// TIA Portal V21 export
FUNCTION "STANDARD" : Void   // FC13, LAD
{ S7_Optimized_Access := 'TRUE' }
// stored: SetENOAutomatically false
   VAR_TEMP
      "std temp3 hyst" : Real;
   END_VAR
   VAR_TEMP   // added for the SCL form of the ladder/FBD networks
      _w1 : Bool;
      _w2 : Bool;
      _w3 : Bool;
      _w4 : Bool;
   END_VAR
BEGIN

REGION Network 1
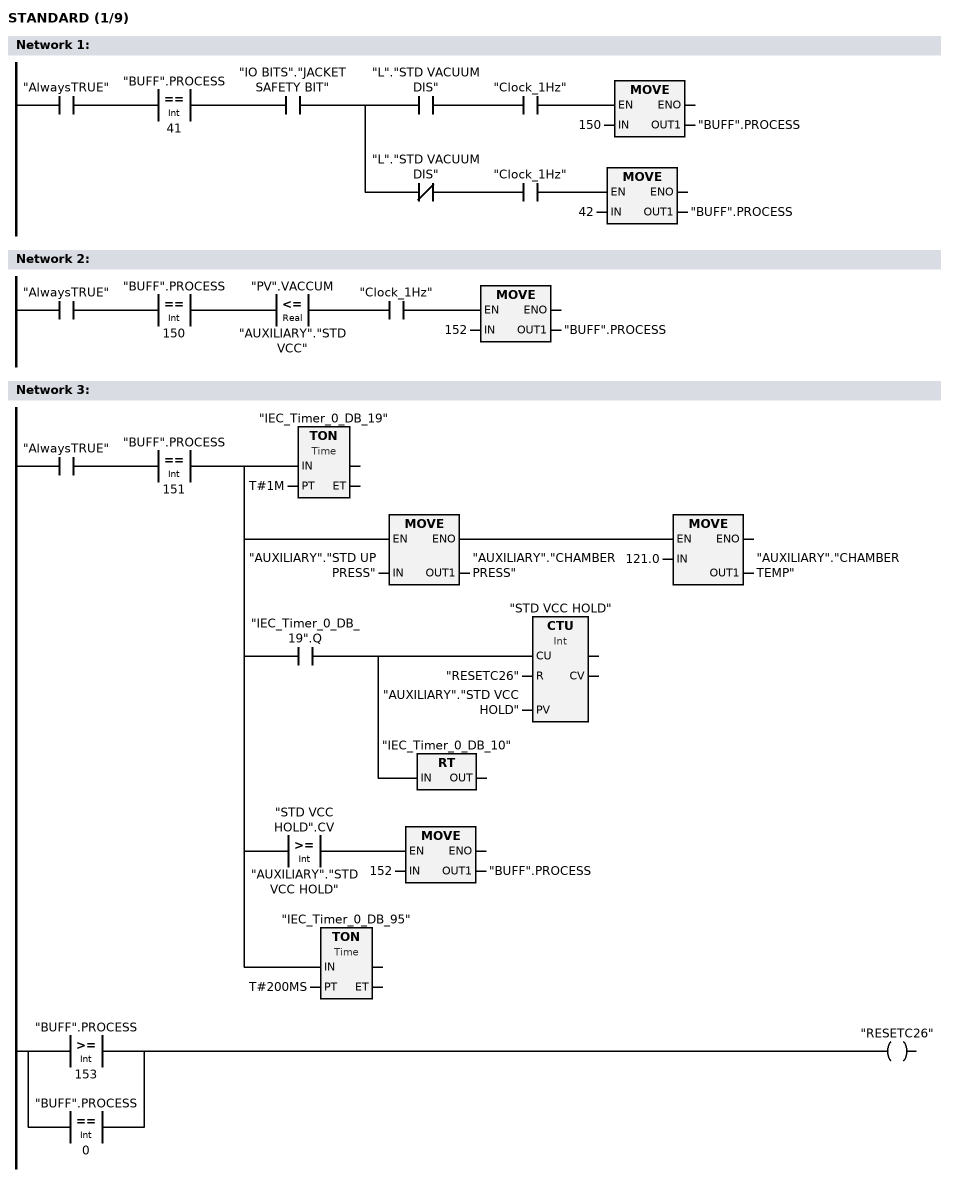
   RUNG wire#powerrail
      Contact( "AlwaysTRUE" )
      { S7_Templates := "SrcType := Int" } EQ_Contact(in1 := "BUFF".PROCESS, in2 := 41)
      Contact( "IO BITS"."JACKET SAFETY BIT" )
      wire#w1
      Contact( "L"."STD VACUUM DIS" )
      Contact( "Clock_1Hz" )
      Move(in := 150, out1 => "BUFF".PROCESS)
   END_RUNG
   RUNG wire#w1
      I_Contact( "L"."STD VACUUM DIS" )
      Contact( "Clock_1Hz" )
      Move(in := 42, out1 => "BUFF".PROCESS)
   END_RUNG
   // the same network as SCL:
   #_w1 := "AlwaysTRUE" AND ("BUFF".PROCESS = 41) AND "IO BITS"."JACKET SAFETY BIT";
   IF #_w1 AND "L"."STD VACUUM DIS" AND "Clock_1Hz" THEN "BUFF".PROCESS := 150; END_IF;
   IF #_w1 AND NOT "L"."STD VACUUM DIS" AND "Clock_1Hz" THEN "BUFF".PROCESS := 42; END_IF;
END_REGION

REGION Network 2
   RUNG wire#powerrail
      Contact( "AlwaysTRUE" )
      { S7_Templates := "SrcType := Int" } EQ_Contact(in1 := "BUFF".PROCESS, in2 := 150)
      { S7_Templates := "SrcType := Real" } LE_Contact(in1 := "PV".VACCUM, in2 := "AUXILIARY"."STD VCC")
      Contact( "Clock_1Hz" )
      Move(in := 152, out1 => "BUFF".PROCESS)
   END_RUNG
   // the same network as SCL:
   IF "AlwaysTRUE" AND ("BUFF".PROCESS = 150) AND ("PV".VACCUM <= "AUXILIARY"."STD VCC") AND "Clock_1Hz" THEN
       "BUFF".PROCESS := 152;
   END_IF;
END_REGION

REGION Network 3
   RUNG wire#powerrail
      Contact( "AlwaysTRUE" )
      { S7_Templates := "SrcType := Int" } EQ_Contact(in1 := "BUFF".PROCESS, in2 := 151)
      wire#w1
      { S7_Templates := "time_type := Time" } "IEC_Timer_0_DB_19".TON(pt := T#1M, et =>)
   END_RUNG
   RUNG wire#w1
      Move(in := "AUXILIARY"."STD UP PRESS", out1 => "AUXILIARY"."CHAMBER PRESS")
      Move(in := 121.0, out1 => "AUXILIARY"."CHAMBER TEMP")
   END_RUNG
   RUNG wire#w1
      Contact( "IEC_Timer_0_DB_19".Q )
      wire#w2
      { S7_Templates := "value_type := Int" } "STD VCC HOLD".CTU(r := "RESETC26", pv := "AUXILIARY"."STD VCC HOLD", cv =>)
   END_RUNG
   RUNG wire#w2
      RT_Coil( "IEC_Timer_0_DB_10" )
   END_RUNG
   RUNG wire#w1
      { S7_Templates := "SrcType := Int" } GE_Contact(in1 := "STD VCC HOLD".CV, in2 := "AUXILIARY"."STD VCC HOLD")
      Move(in := 152, out1 => "BUFF".PROCESS)
   END_RUNG
   RUNG wire#w1
      { S7_Templates := "time_type := Time" } "IEC_Timer_0_DB_95".TON(pt := T#200MS, et =>)
   END_RUNG
   RUNG wire#powerrail
      { S7_Templates := "SrcType := Int" } GE_Contact(in1 := "BUFF".PROCESS, in2 := 153)
      wire#w3
      Coil( "RESETC26" )
   END_RUNG
   RUNG wire#powerrail
      { S7_Templates := "SrcType := Int" } EQ_Contact(in1 := "BUFF".PROCESS, in2 := 0)
   END_RUNG wire#w3
   // the same network as SCL:
   #_w1 := "AlwaysTRUE" AND ("BUFF".PROCESS = 151);
   "IEC_Timer_0_DB_19".TON(IN := #_w1, PT := T#1M);
   IF #_w1 THEN
       "AUXILIARY"."CHAMBER PRESS" := "AUXILIARY"."STD UP PRESS";
       "AUXILIARY"."CHAMBER TEMP" := 121.0;
   END_IF;
   #_w2 := #_w1 AND "IEC_Timer_0_DB_19".Q;
   "STD VCC HOLD".CTU(CU := #_w2, R := "RESETC26", PV := "AUXILIARY"."STD VCC HOLD");
   IF #_w2 THEN RESET_TIMER("IEC_Timer_0_DB_10"); END_IF;
   IF #_w1 AND ("STD VCC HOLD".CV >= "AUXILIARY"."STD VCC HOLD") THEN "BUFF".PROCESS := 152; END_IF;
   "IEC_Timer_0_DB_95".TON(IN := #_w1, PT := T#200MS);
   "RESETC26" := ("BUFF".PROCESS >= 153) OR ("BUFF".PROCESS = 0);
END_REGION

REGION Network 4
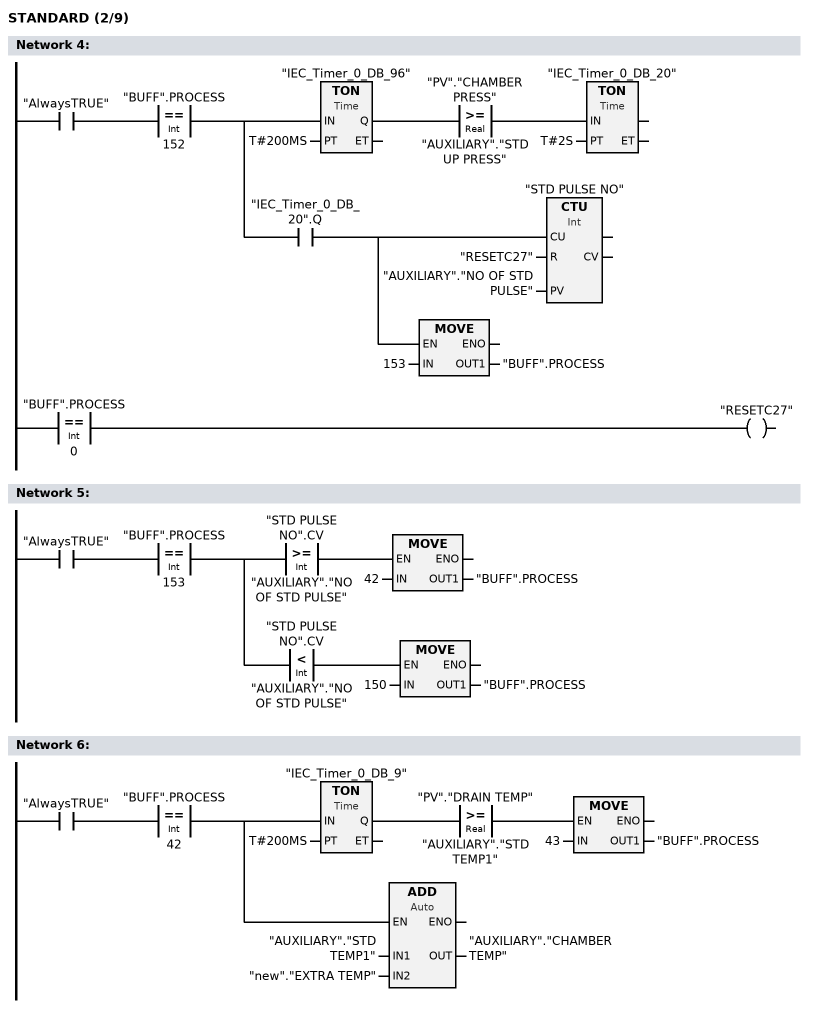
   RUNG wire#powerrail
      Contact( "AlwaysTRUE" )
      { S7_Templates := "SrcType := Int" } EQ_Contact(in1 := "BUFF".PROCESS, in2 := 152)
      wire#w1
      { S7_Templates := "time_type := Time" } "IEC_Timer_0_DB_96".TON(pt := T#200MS, et =>)
      { S7_Templates := "SrcType := Real" } GE_Contact(in1 := "PV"."CHAMBER PRESS", in2 := "AUXILIARY"."STD UP PRESS")
      { S7_Templates := "time_type := Time" } "IEC_Timer_0_DB_20".TON(pt := T#2S, et =>)
   END_RUNG
   RUNG wire#w1
      Contact( "IEC_Timer_0_DB_20".Q )
      wire#w2
      { S7_Templates := "value_type := Int" } "STD PULSE NO".CTU(r := "RESETC27", pv := "AUXILIARY"."NO OF STD PULSE", cv =>)
   END_RUNG
   RUNG wire#w2
      Move(in := 153, out1 => "BUFF".PROCESS)
   END_RUNG
   RUNG wire#powerrail
      { S7_Templates := "SrcType := Int" } EQ_Contact(in1 := "BUFF".PROCESS, in2 := 0)
      Coil( "RESETC27" )
   END_RUNG
   // the same network as SCL:
   #_w1 := "AlwaysTRUE" AND ("BUFF".PROCESS = 152);
   "IEC_Timer_0_DB_96".TON(IN := #_w1, PT := T#200MS);
   "IEC_Timer_0_DB_20".TON(IN := "IEC_Timer_0_DB_96".Q AND ("PV"."CHAMBER PRESS" >= "AUXILIARY"."STD UP PRESS"),
                           PT := T#2S);
   #_w2 := #_w1 AND "IEC_Timer_0_DB_20".Q;
   "STD PULSE NO".CTU(CU := #_w2, R := "RESETC27", PV := "AUXILIARY"."NO OF STD PULSE");
   IF #_w2 THEN "BUFF".PROCESS := 153; END_IF;
   "RESETC27" := "BUFF".PROCESS = 0;
END_REGION

REGION Network 5
   RUNG wire#powerrail
      Contact( "AlwaysTRUE" )
      { S7_Templates := "SrcType := Int" } EQ_Contact(in1 := "BUFF".PROCESS, in2 := 153)
      wire#w1
      { S7_Templates := "SrcType := Int" } GE_Contact(in1 := "STD PULSE NO".CV, in2 := "AUXILIARY"."NO OF STD PULSE")
      Move(in := 42, out1 => "BUFF".PROCESS)
   END_RUNG
   RUNG wire#w1
      { S7_Templates := "SrcType := Int" } LT_Contact(in1 := "STD PULSE NO".CV, in2 := "AUXILIARY"."NO OF STD PULSE")
      Move(in := 150, out1 => "BUFF".PROCESS)
   END_RUNG
   // the same network as SCL:
   #_w1 := "AlwaysTRUE" AND ("BUFF".PROCESS = 153);
   IF #_w1 AND ("STD PULSE NO".CV >= "AUXILIARY"."NO OF STD PULSE") THEN "BUFF".PROCESS := 42; END_IF;
   IF #_w1 AND ("STD PULSE NO".CV < "AUXILIARY"."NO OF STD PULSE") THEN "BUFF".PROCESS := 150; END_IF;
END_REGION

REGION Network 6
   RUNG wire#powerrail
      Contact( "AlwaysTRUE" )
      { S7_Templates := "SrcType := Int" } EQ_Contact(in1 := "BUFF".PROCESS, in2 := 42)
      wire#w1
      { S7_Templates := "time_type := Time" } "IEC_Timer_0_DB_9".TON(pt := T#200MS, et =>)
      { S7_Templates := "SrcType := Real" } GE_Contact(in1 := "PV"."DRAIN TEMP", in2 := "AUXILIARY"."STD TEMP1")
      Move(in := 43, out1 => "BUFF".PROCESS)
   END_RUNG
   RUNG wire#w1
      Add(in1 := "AUXILIARY"."STD TEMP1", in2 := "new"."EXTRA TEMP", out => "AUXILIARY"."CHAMBER TEMP")
   END_RUNG
   // the same network as SCL:
   #_w1 := "AlwaysTRUE" AND ("BUFF".PROCESS = 42);
   "IEC_Timer_0_DB_9".TON(IN := #_w1, PT := T#200MS);
   IF "IEC_Timer_0_DB_9".Q AND ("PV"."DRAIN TEMP" >= "AUXILIARY"."STD TEMP1") THEN
       "BUFF".PROCESS := 43;
   END_IF;
   IF #_w1 THEN "AUXILIARY"."CHAMBER TEMP" := "AUXILIARY"."STD TEMP1" + "new"."EXTRA TEMP"; END_IF;
END_REGION

REGION Network 7
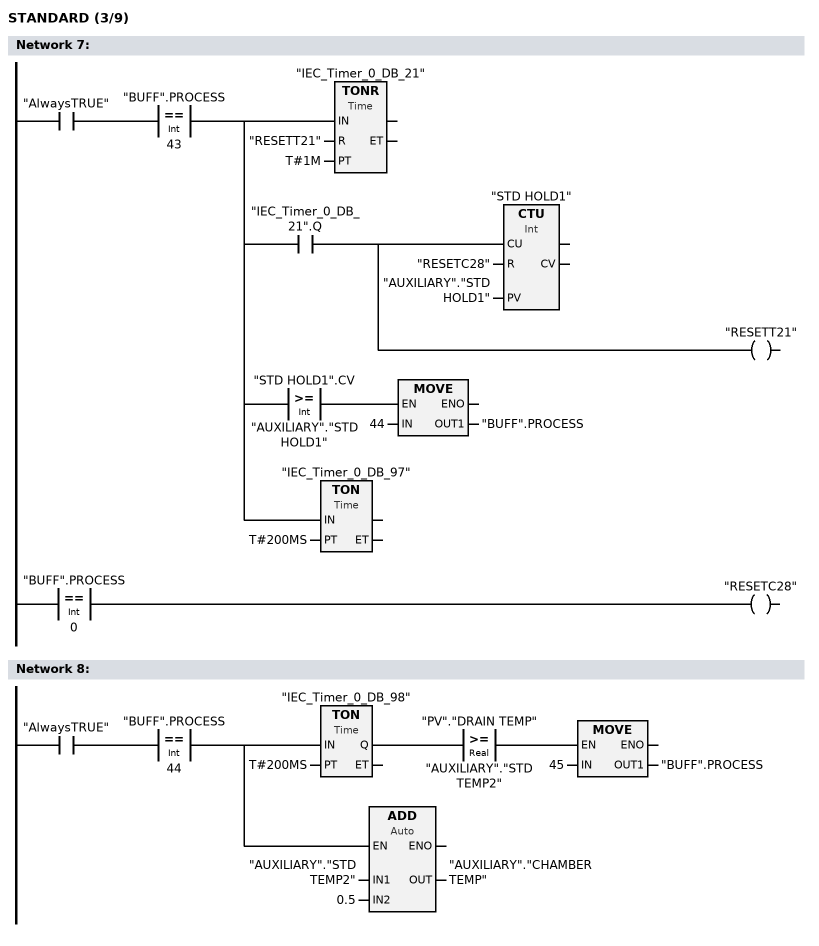
   RUNG wire#powerrail
      Contact( "AlwaysTRUE" )
      { S7_Templates := "SrcType := Int" } EQ_Contact(in1 := "BUFF".PROCESS, in2 := 43)
      wire#w1
      { S7_Templates := "time_type := Time" } "IEC_Timer_0_DB_21".TONR(r := "RESETT21", pt := T#1M, et =>)
   END_RUNG
   RUNG wire#w1
      Contact( "IEC_Timer_0_DB_21".Q )
      wire#w2
      { S7_Templates := "value_type := Int" } "STD HOLD1".CTU(r := "RESETC28", pv := "AUXILIARY"."STD HOLD1", cv =>)
   END_RUNG
   RUNG wire#w2
      Coil( "RESETT21" )
   END_RUNG
   RUNG wire#w1
      { S7_Templates := "SrcType := Int" } GE_Contact(in1 := "STD HOLD1".CV, in2 := "AUXILIARY"."STD HOLD1")
      Move(in := 44, out1 => "BUFF".PROCESS)
   END_RUNG
   RUNG wire#w1
      { S7_Templates := "time_type := Time" } "IEC_Timer_0_DB_97".TON(pt := T#200MS, et =>)
   END_RUNG
   RUNG wire#powerrail
      { S7_Templates := "SrcType := Int" } EQ_Contact(in1 := "BUFF".PROCESS, in2 := 0)
      Coil( "RESETC28" )
   END_RUNG
   // the same network as SCL:
   #_w1 := "AlwaysTRUE" AND ("BUFF".PROCESS = 43);
   "IEC_Timer_0_DB_21".TONR(IN := #_w1, R := "RESETT21", PT := T#1M);
   #_w2 := #_w1 AND "IEC_Timer_0_DB_21".Q;
   "STD HOLD1".CTU(CU := #_w2, R := "RESETC28", PV := "AUXILIARY"."STD HOLD1");
   "RESETT21" := #_w2;
   IF #_w1 AND ("STD HOLD1".CV >= "AUXILIARY"."STD HOLD1") THEN "BUFF".PROCESS := 44; END_IF;
   "IEC_Timer_0_DB_97".TON(IN := #_w1, PT := T#200MS);
   "RESETC28" := "BUFF".PROCESS = 0;
END_REGION

REGION Network 8
   RUNG wire#powerrail
      Contact( "AlwaysTRUE" )
      { S7_Templates := "SrcType := Int" } EQ_Contact(in1 := "BUFF".PROCESS, in2 := 44)
      wire#w1
      { S7_Templates := "time_type := Time" } "IEC_Timer_0_DB_98".TON(pt := T#200MS, et =>)
      { S7_Templates := "SrcType := Real" } GE_Contact(in1 := "PV"."DRAIN TEMP", in2 := "AUXILIARY"."STD TEMP2")
      Move(in := 45, out1 => "BUFF".PROCESS)
   END_RUNG
   RUNG wire#w1
      Add(in1 := "AUXILIARY"."STD TEMP2", in2 := 0.5, out => "AUXILIARY"."CHAMBER TEMP")
   END_RUNG
   // the same network as SCL:
   #_w1 := "AlwaysTRUE" AND ("BUFF".PROCESS = 44);
   "IEC_Timer_0_DB_98".TON(IN := #_w1, PT := T#200MS);
   IF "IEC_Timer_0_DB_98".Q AND ("PV"."DRAIN TEMP" >= "AUXILIARY"."STD TEMP2") THEN
       "BUFF".PROCESS := 45;
   END_IF;
   IF #_w1 THEN "AUXILIARY"."CHAMBER TEMP" := "AUXILIARY"."STD TEMP2" + 0.5; END_IF;
END_REGION

REGION Network 9
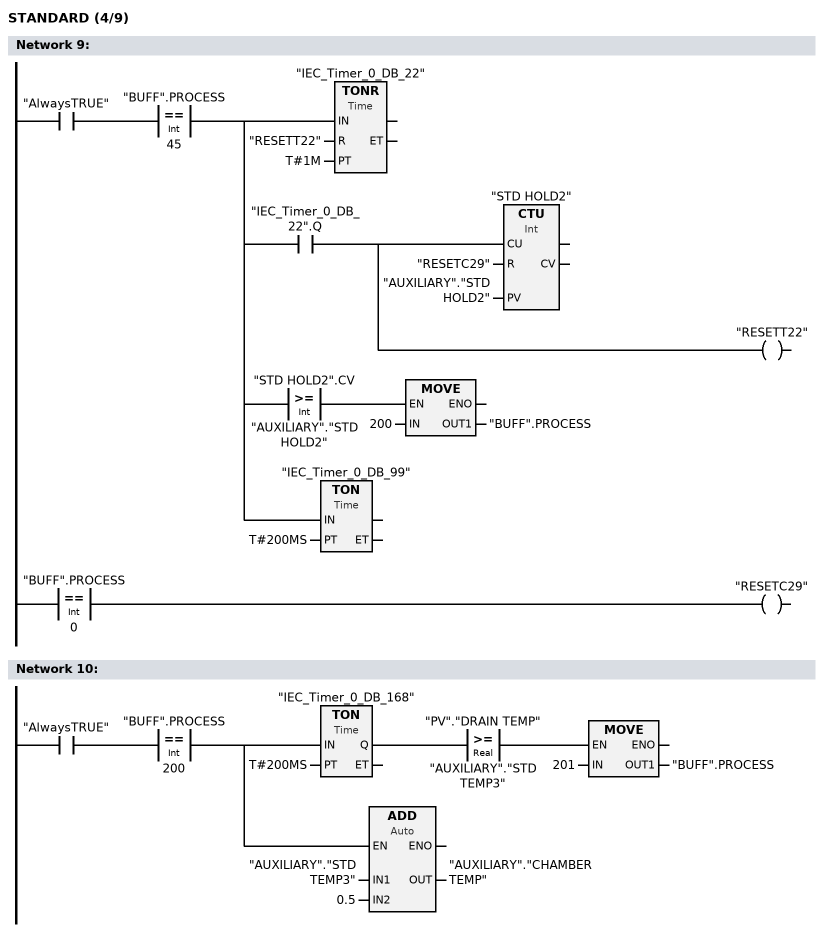
   RUNG wire#powerrail
      Contact( "AlwaysTRUE" )
      { S7_Templates := "SrcType := Int" } EQ_Contact(in1 := "BUFF".PROCESS, in2 := 45)
      wire#w1
      { S7_Templates := "time_type := Time" } "IEC_Timer_0_DB_22".TONR(r := "RESETT22", pt := T#1M, et =>)
   END_RUNG
   RUNG wire#w1
      Contact( "IEC_Timer_0_DB_22".Q )
      wire#w2
      { S7_Templates := "value_type := Int" } "STD HOLD2".CTU(r := "RESETC29", pv := "AUXILIARY"."STD HOLD2", cv =>)
   END_RUNG
   RUNG wire#w2
      Coil( "RESETT22" )
   END_RUNG
   RUNG wire#w1
      { S7_Templates := "SrcType := Int" } GE_Contact(in1 := "STD HOLD2".CV, in2 := "AUXILIARY"."STD HOLD2")
      Move(in := 200, out1 => "BUFF".PROCESS)
   END_RUNG
   RUNG wire#w1
      { S7_Templates := "time_type := Time" } "IEC_Timer_0_DB_99".TON(pt := T#200MS, et =>)
   END_RUNG
   RUNG wire#powerrail
      { S7_Templates := "SrcType := Int" } EQ_Contact(in1 := "BUFF".PROCESS, in2 := 0)
      Coil( "RESETC29" )
   END_RUNG
   // the same network as SCL:
   #_w1 := "AlwaysTRUE" AND ("BUFF".PROCESS = 45);
   "IEC_Timer_0_DB_22".TONR(IN := #_w1, R := "RESETT22", PT := T#1M);
   #_w2 := #_w1 AND "IEC_Timer_0_DB_22".Q;
   "STD HOLD2".CTU(CU := #_w2, R := "RESETC29", PV := "AUXILIARY"."STD HOLD2");
   "RESETT22" := #_w2;
   IF #_w1 AND ("STD HOLD2".CV >= "AUXILIARY"."STD HOLD2") THEN "BUFF".PROCESS := 200; END_IF;
   "IEC_Timer_0_DB_99".TON(IN := #_w1, PT := T#200MS);
   "RESETC29" := "BUFF".PROCESS = 0;
END_REGION

REGION Network 10
   RUNG wire#powerrail
      Contact( "AlwaysTRUE" )
      { S7_Templates := "SrcType := Int" } EQ_Contact(in1 := "BUFF".PROCESS, in2 := 200)
      wire#w1
      { S7_Templates := "time_type := Time" } "IEC_Timer_0_DB_168".TON(pt := T#200MS, et =>)
      { S7_Templates := "SrcType := Real" } GE_Contact(in1 := "PV"."DRAIN TEMP", in2 := "AUXILIARY"."STD TEMP3")
      Move(in := 201, out1 => "BUFF".PROCESS)
   END_RUNG
   RUNG wire#w1
      Add(in1 := "AUXILIARY"."STD TEMP3", in2 := 0.5, out => "AUXILIARY"."CHAMBER TEMP")
   END_RUNG
   // the same network as SCL:
   #_w1 := "AlwaysTRUE" AND ("BUFF".PROCESS = 200);
   "IEC_Timer_0_DB_168".TON(IN := #_w1, PT := T#200MS);
   IF "IEC_Timer_0_DB_168".Q AND ("PV"."DRAIN TEMP" >= "AUXILIARY"."STD TEMP3") THEN
       "BUFF".PROCESS := 201;
   END_IF;
   IF #_w1 THEN "AUXILIARY"."CHAMBER TEMP" := "AUXILIARY"."STD TEMP3" + 0.5; END_IF;
END_REGION

REGION Network 11
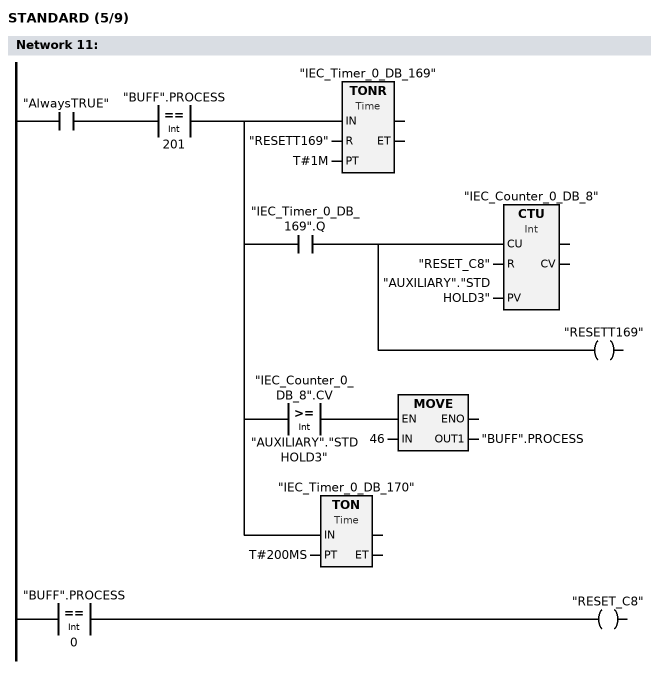
   RUNG wire#powerrail
      Contact( "AlwaysTRUE" )
      { S7_Templates := "SrcType := Int" } EQ_Contact(in1 := "BUFF".PROCESS, in2 := 201)
      wire#w1
      { S7_Templates := "time_type := Time" } "IEC_Timer_0_DB_169".TONR(r := "RESETT169", pt := T#1M, et =>)
   END_RUNG
   RUNG wire#w1
      Contact( "IEC_Timer_0_DB_169".Q )
      wire#w2
      { S7_Templates := "value_type := Int" } "IEC_Counter_0_DB_8".CTU(r := "RESET_C8", pv := "AUXILIARY"."STD HOLD3", cv =>)
   END_RUNG
   RUNG wire#w2
      Coil( "RESETT169" )
   END_RUNG
   RUNG wire#w1
      { S7_Templates := "SrcType := Int" } GE_Contact(in1 := "IEC_Counter_0_DB_8".CV, in2 := "AUXILIARY"."STD HOLD3")
      Move(in := 46, out1 => "BUFF".PROCESS)
   END_RUNG
   RUNG wire#w1
      { S7_Templates := "time_type := Time" } "IEC_Timer_0_DB_170".TON(pt := T#200MS, et =>)
   END_RUNG
   RUNG wire#powerrail
      { S7_Templates := "SrcType := Int" } EQ_Contact(in1 := "BUFF".PROCESS, in2 := 0)
      Coil( "RESET_C8" )
   END_RUNG
   // the same network as SCL:
   #_w1 := "AlwaysTRUE" AND ("BUFF".PROCESS = 201);
   "IEC_Timer_0_DB_169".TONR(IN := #_w1, R := "RESETT169", PT := T#1M);
   #_w2 := #_w1 AND "IEC_Timer_0_DB_169".Q;
   "IEC_Counter_0_DB_8".CTU(CU := #_w2, R := "RESET_C8", PV := "AUXILIARY"."STD HOLD3");
   "RESETT169" := #_w2;
   IF #_w1 AND ("IEC_Counter_0_DB_8".CV >= "AUXILIARY"."STD HOLD3") THEN "BUFF".PROCESS := 46; END_IF;
   "IEC_Timer_0_DB_170".TON(IN := #_w1, PT := T#200MS);
   "RESET_C8" := "BUFF".PROCESS = 0;
END_REGION

REGION Network 12
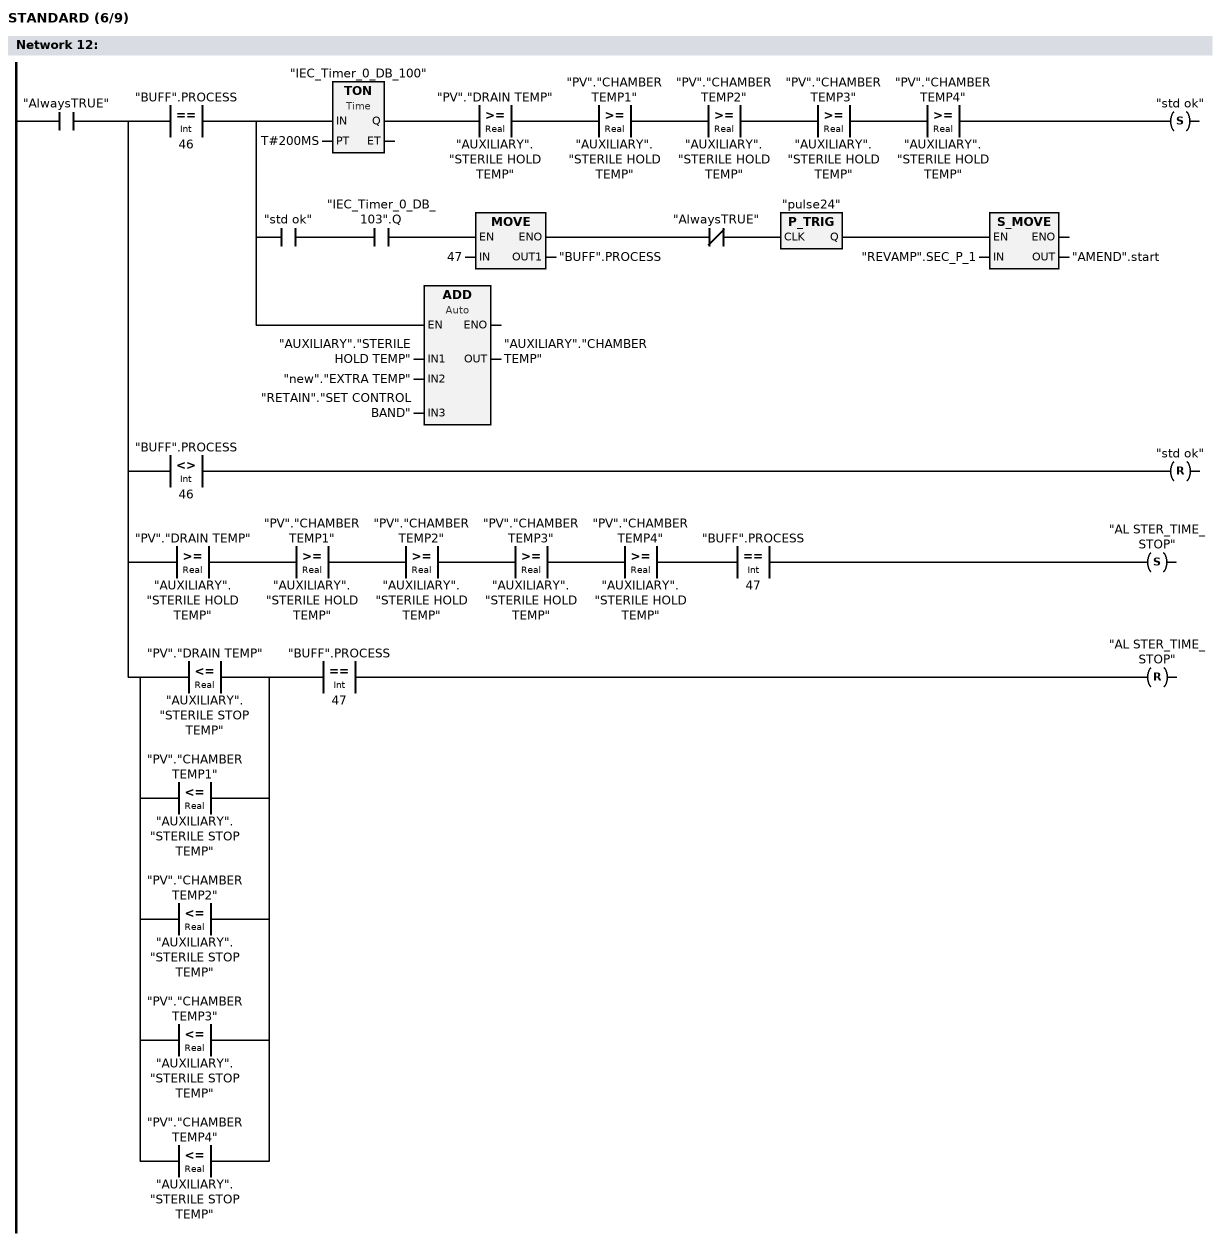
   RUNG wire#powerrail
      Contact( "AlwaysTRUE" )
      wire#w1
      { S7_Templates := "SrcType := Int" } EQ_Contact(in1 := "BUFF".PROCESS, in2 := 46)
      wire#w2
      { S7_Templates := "time_type := Time" } "IEC_Timer_0_DB_100".TON(pt := T#200MS, et =>)
      { S7_Templates := "SrcType := Real" } GE_Contact(in1 := "PV"."DRAIN TEMP", in2 := "AUXILIARY"."STERILE HOLD TEMP")
      { S7_Templates := "SrcType := Real" } GE_Contact(in1 := "PV"."CHAMBER TEMP1", in2 := "AUXILIARY"."STERILE HOLD TEMP")
      { S7_Templates := "SrcType := Real" } GE_Contact(in1 := "PV"."CHAMBER TEMP2", in2 := "AUXILIARY"."STERILE HOLD TEMP")
      { S7_Templates := "SrcType := Real" } GE_Contact(in1 := "PV"."CHAMBER TEMP3", in2 := "AUXILIARY"."STERILE HOLD TEMP")
      { S7_Templates := "SrcType := Real" } GE_Contact(in1 := "PV"."CHAMBER TEMP4", in2 := "AUXILIARY"."STERILE HOLD TEMP")
      S_Coil( "std ok" )
   END_RUNG
   RUNG wire#w2
      Contact( "std ok" )
      Contact( "IEC_Timer_0_DB_103".Q )
      Move(in := 47, out1 => "BUFF".PROCESS)
      I_Contact( "AlwaysTRUE" )
      P_Trig( "pulse24" )
      S_Move(in := "REVAMP".SEC_P_1, out => "AMEND".start)
   END_RUNG
   RUNG wire#w2
      Add(in1 := "AUXILIARY"."STERILE HOLD TEMP", in2 := "new"."EXTRA TEMP", in3 := "RETAIN"."SET CONTROL BAND", out => "AUXILIARY"."CHAMBER TEMP")
   END_RUNG
   RUNG wire#w1
      { S7_Templates := "SrcType := Int" } NE_Contact(in1 := "BUFF".PROCESS, in2 := 46)
      R_Coil( "std ok" )
   END_RUNG
   RUNG wire#w1
      { S7_Templates := "SrcType := Real" } GE_Contact(in1 := "PV"."DRAIN TEMP", in2 := "AUXILIARY"."STERILE HOLD TEMP")
      { S7_Templates := "SrcType := Real" } GE_Contact(in1 := "PV"."CHAMBER TEMP1", in2 := "AUXILIARY"."STERILE HOLD TEMP")
      { S7_Templates := "SrcType := Real" } GE_Contact(in1 := "PV"."CHAMBER TEMP2", in2 := "AUXILIARY"."STERILE HOLD TEMP")
      { S7_Templates := "SrcType := Real" } GE_Contact(in1 := "PV"."CHAMBER TEMP3", in2 := "AUXILIARY"."STERILE HOLD TEMP")
      { S7_Templates := "SrcType := Real" } GE_Contact(in1 := "PV"."CHAMBER TEMP4", in2 := "AUXILIARY"."STERILE HOLD TEMP")
      { S7_Templates := "SrcType := Int" } EQ_Contact(in1 := "BUFF".PROCESS, in2 := 47)
      S_Coil( "AL STER_TIME_STOP" )
   END_RUNG
   RUNG wire#w1
      { S7_Templates := "SrcType := Real" } LE_Contact(in1 := "PV"."DRAIN TEMP", in2 := "AUXILIARY"."STERILE STOP TEMP")
      wire#w3
      { S7_Templates := "SrcType := Int" } EQ_Contact(in1 := "BUFF".PROCESS, in2 := 47)
      R_Coil( "AL STER_TIME_STOP" )
   END_RUNG
   RUNG wire#w1
      { S7_Templates := "SrcType := Real" } LE_Contact(in1 := "PV"."CHAMBER TEMP1", in2 := "AUXILIARY"."STERILE STOP TEMP")
   END_RUNG wire#w3
   RUNG wire#w1
      { S7_Templates := "SrcType := Real" } LE_Contact(in1 := "PV"."CHAMBER TEMP2", in2 := "AUXILIARY"."STERILE STOP TEMP")
   END_RUNG wire#w3
   RUNG wire#w1
      { S7_Templates := "SrcType := Real" } LE_Contact(in1 := "PV"."CHAMBER TEMP3", in2 := "AUXILIARY"."STERILE STOP TEMP")
   END_RUNG wire#w3
   RUNG wire#w1
      { S7_Templates := "SrcType := Real" } LE_Contact(in1 := "PV"."CHAMBER TEMP4", in2 := "AUXILIARY"."STERILE STOP TEMP")
   END_RUNG wire#w3
   // the same network as SCL:
   #_w1 := "AlwaysTRUE" AND ("BUFF".PROCESS = 46);
   "IEC_Timer_0_DB_100".TON(IN := #_w1, PT := T#200MS);
   IF "IEC_Timer_0_DB_100".Q AND ("PV"."DRAIN TEMP" >= "AUXILIARY"."STERILE HOLD TEMP") AND ("PV"."CHAMBER TEMP1" >= "AUXILIARY"."STERILE HOLD TEMP") AND ("PV"."CHAMBER TEMP2" >= "AUXILIARY"."STERILE HOLD TEMP") AND ("PV"."CHAMBER TEMP3" >= "AUXILIARY"."STERILE HOLD TEMP") AND ("PV"."CHAMBER TEMP4" >= "AUXILIARY"."STERILE HOLD TEMP") THEN
       "std ok" := TRUE;
   END_IF;
   #_w2 := #_w1 AND "std ok" AND "IEC_Timer_0_DB_103".Q;
   IF #_w2 THEN "BUFF".PROCESS := 47; END_IF;
   #_w3 := #_w2 AND NOT "AlwaysTRUE";
   #_w4 := #_w3 AND NOT "pulse24";   // rising edge
   "pulse24" := #_w3;
   IF #_w4 THEN "AMEND".start := "REVAMP".SEC_P_1; END_IF;
   IF #_w1 THEN
       "AUXILIARY"."CHAMBER TEMP" := "AUXILIARY"."STERILE HOLD TEMP" + "new"."EXTRA TEMP" + "RETAIN"."SET CONTROL BAND";
   END_IF;
   IF "AlwaysTRUE" AND ("BUFF".PROCESS <> 46) THEN "std ok" := FALSE; END_IF;
   IF "AlwaysTRUE" AND ("PV"."DRAIN TEMP" >= "AUXILIARY"."STERILE HOLD TEMP") AND ("PV"."CHAMBER TEMP1" >= "AUXILIARY"."STERILE HOLD TEMP") AND ("PV"."CHAMBER TEMP2" >= "AUXILIARY"."STERILE HOLD TEMP") AND ("PV"."CHAMBER TEMP3" >= "AUXILIARY"."STERILE HOLD TEMP") AND ("PV"."CHAMBER TEMP4" >= "AUXILIARY"."STERILE HOLD TEMP") AND ("BUFF".PROCESS = 47) THEN
       "AL STER_TIME_STOP" := TRUE;
   END_IF;
   IF "AlwaysTRUE" AND (("PV"."DRAIN TEMP" <= "AUXILIARY"."STERILE STOP TEMP") OR ("PV"."CHAMBER TEMP1" <= "AUXILIARY"."STERILE STOP TEMP") OR ("PV"."CHAMBER TEMP2" <= "AUXILIARY"."STERILE STOP TEMP") OR ("PV"."CHAMBER TEMP3" <= "AUXILIARY"."STERILE STOP TEMP") OR ("PV"."CHAMBER TEMP4" <= "AUXILIARY"."STERILE STOP TEMP")) AND ("BUFF".PROCESS = 47) THEN
       "AL STER_TIME_STOP" := FALSE;
   END_IF;
END_REGION

REGION Network 13
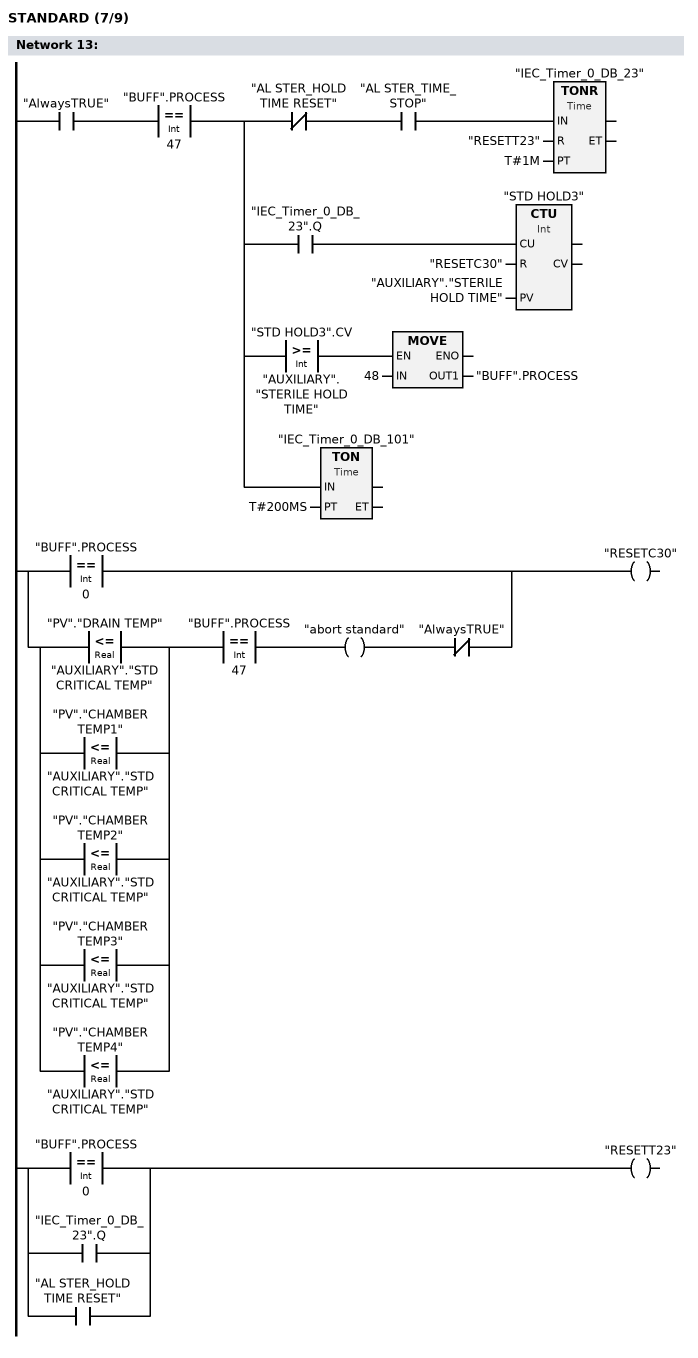
   RUNG wire#powerrail
      Contact( "AlwaysTRUE" )
      { S7_Templates := "SrcType := Int" } EQ_Contact(in1 := "BUFF".PROCESS, in2 := 47)
      wire#w1
      I_Contact( "AL STER_HOLD TIME RESET" )
      Contact( "AL STER_TIME_STOP" )
      { S7_Templates := "time_type := Time" } "IEC_Timer_0_DB_23".TONR(r := "RESETT23", pt := T#1M, et =>)
   END_RUNG
   RUNG wire#w1
      Contact( "IEC_Timer_0_DB_23".Q )
      { S7_Templates := "value_type := Int" } "STD HOLD3".CTU(r := "RESETC30", pv := "AUXILIARY"."STERILE HOLD TIME", cv =>)
   END_RUNG
   RUNG wire#w1
      { S7_Templates := "SrcType := Int" } GE_Contact(in1 := "STD HOLD3".CV, in2 := "AUXILIARY"."STERILE HOLD TIME")
      Move(in := 48, out1 => "BUFF".PROCESS)
   END_RUNG
   RUNG wire#w1
      { S7_Templates := "time_type := Time" } "IEC_Timer_0_DB_101".TON(pt := T#200MS, et =>)
   END_RUNG
   RUNG wire#powerrail
      { S7_Templates := "SrcType := Int" } EQ_Contact(in1 := "BUFF".PROCESS, in2 := 0)
      wire#w2
      Coil( "RESETC30" )
   END_RUNG
   RUNG wire#powerrail
      { S7_Templates := "SrcType := Real" } LE_Contact(in1 := "PV"."DRAIN TEMP", in2 := "AUXILIARY"."STD CRITICAL TEMP")
      wire#w3
      { S7_Templates := "SrcType := Int" } EQ_Contact(in1 := "BUFF".PROCESS, in2 := 47)
      Coil( "abort standard" )
      I_Contact( "AlwaysTRUE" )
   END_RUNG wire#w2
   RUNG wire#powerrail
      { S7_Templates := "SrcType := Real" } LE_Contact(in1 := "PV"."CHAMBER TEMP1", in2 := "AUXILIARY"."STD CRITICAL TEMP")
   END_RUNG wire#w3
   RUNG wire#powerrail
      { S7_Templates := "SrcType := Real" } LE_Contact(in1 := "PV"."CHAMBER TEMP2", in2 := "AUXILIARY"."STD CRITICAL TEMP")
   END_RUNG wire#w3
   RUNG wire#powerrail
      { S7_Templates := "SrcType := Real" } LE_Contact(in1 := "PV"."CHAMBER TEMP3", in2 := "AUXILIARY"."STD CRITICAL TEMP")
   END_RUNG wire#w3
   RUNG wire#powerrail
      { S7_Templates := "SrcType := Real" } LE_Contact(in1 := "PV"."CHAMBER TEMP4", in2 := "AUXILIARY"."STD CRITICAL TEMP")
   END_RUNG wire#w3
   RUNG wire#powerrail
      { S7_Templates := "SrcType := Int" } EQ_Contact(in1 := "BUFF".PROCESS, in2 := 0)
      wire#w4
      Coil( "RESETT23" )
   END_RUNG
   RUNG wire#powerrail
      Contact( "IEC_Timer_0_DB_23".Q )
   END_RUNG wire#w4
   RUNG wire#powerrail
      Contact( "AL STER_HOLD TIME RESET" )
   END_RUNG wire#w4
   // the same network as SCL:
   #_w1 := "AlwaysTRUE" AND ("BUFF".PROCESS = 47);
   "IEC_Timer_0_DB_23".TONR(IN := #_w1 AND NOT "AL STER_HOLD TIME RESET" AND "AL STER_TIME_STOP",
                           R := "RESETT23",
                           PT := T#1M);
   "STD HOLD3".CTU(CU := #_w1 AND "IEC_Timer_0_DB_23".Q, R := "RESETC30", PV := "AUXILIARY"."STERILE HOLD TIME");
   IF #_w1 AND ("STD HOLD3".CV >= "AUXILIARY"."STERILE HOLD TIME") THEN "BUFF".PROCESS := 48; END_IF;
   "IEC_Timer_0_DB_101".TON(IN := #_w1, PT := T#200MS);
   "abort standard" := (("PV"."DRAIN TEMP" <= "AUXILIARY"."STD CRITICAL TEMP") OR ("PV"."CHAMBER TEMP1" <= "AUXILIARY"."STD CRITICAL TEMP") OR ("PV"."CHAMBER TEMP2" <= "AUXILIARY"."STD CRITICAL TEMP") OR ("PV"."CHAMBER TEMP3" <= "AUXILIARY"."STD CRITICAL TEMP") OR ("PV"."CHAMBER TEMP4" <= "AUXILIARY"."STD CRITICAL TEMP")) AND ("BUFF".PROCESS = 47);
   "RESETC30" := ("BUFF".PROCESS = 0) OR ("abort standard" AND NOT "AlwaysTRUE");
   "RESETT23" := ("BUFF".PROCESS = 0) OR "IEC_Timer_0_DB_23".Q OR "AL STER_HOLD TIME RESET";
END_REGION

REGION Network 14
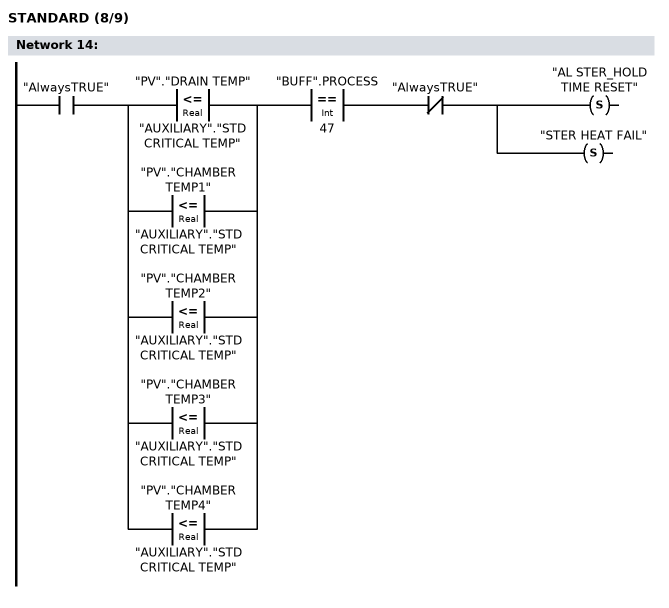
   RUNG wire#powerrail
      Contact( "AlwaysTRUE" )
      wire#w1
      { S7_Templates := "SrcType := Real" } LE_Contact(in1 := "PV"."DRAIN TEMP", in2 := "AUXILIARY"."STD CRITICAL TEMP")
      wire#w2
      { S7_Templates := "SrcType := Int" } EQ_Contact(in1 := "BUFF".PROCESS, in2 := 47)
      I_Contact( "AlwaysTRUE" )
      wire#w3
      S_Coil( "AL STER_HOLD TIME RESET" )
   END_RUNG
   RUNG wire#w1
      { S7_Templates := "SrcType := Real" } LE_Contact(in1 := "PV"."CHAMBER TEMP1", in2 := "AUXILIARY"."STD CRITICAL TEMP")
   END_RUNG wire#w2
   RUNG wire#w1
      { S7_Templates := "SrcType := Real" } LE_Contact(in1 := "PV"."CHAMBER TEMP2", in2 := "AUXILIARY"."STD CRITICAL TEMP")
   END_RUNG wire#w2
   RUNG wire#w1
      { S7_Templates := "SrcType := Real" } LE_Contact(in1 := "PV"."CHAMBER TEMP3", in2 := "AUXILIARY"."STD CRITICAL TEMP")
   END_RUNG wire#w2
   RUNG wire#w1
      { S7_Templates := "SrcType := Real" } LE_Contact(in1 := "PV"."CHAMBER TEMP4", in2 := "AUXILIARY"."STD CRITICAL TEMP")
   END_RUNG wire#w2
   RUNG wire#w3
      S_Coil( "STER HEAT FAIL" )
   END_RUNG
   // the same network as SCL:
   IF "AlwaysTRUE" AND (("PV"."DRAIN TEMP" <= "AUXILIARY"."STD CRITICAL TEMP") OR ("PV"."CHAMBER TEMP1" <= "AUXILIARY"."STD CRITICAL TEMP") OR ("PV"."CHAMBER TEMP2" <= "AUXILIARY"."STD CRITICAL TEMP") OR ("PV"."CHAMBER TEMP3" <= "AUXILIARY"."STD CRITICAL TEMP") OR ("PV"."CHAMBER TEMP4" <= "AUXILIARY"."STD CRITICAL TEMP")) AND ("BUFF".PROCESS = 47) AND NOT "AlwaysTRUE" THEN
       "AL STER_HOLD TIME RESET" := TRUE;
       "STER HEAT FAIL" := TRUE;
   END_IF;
END_REGION

REGION Network 15
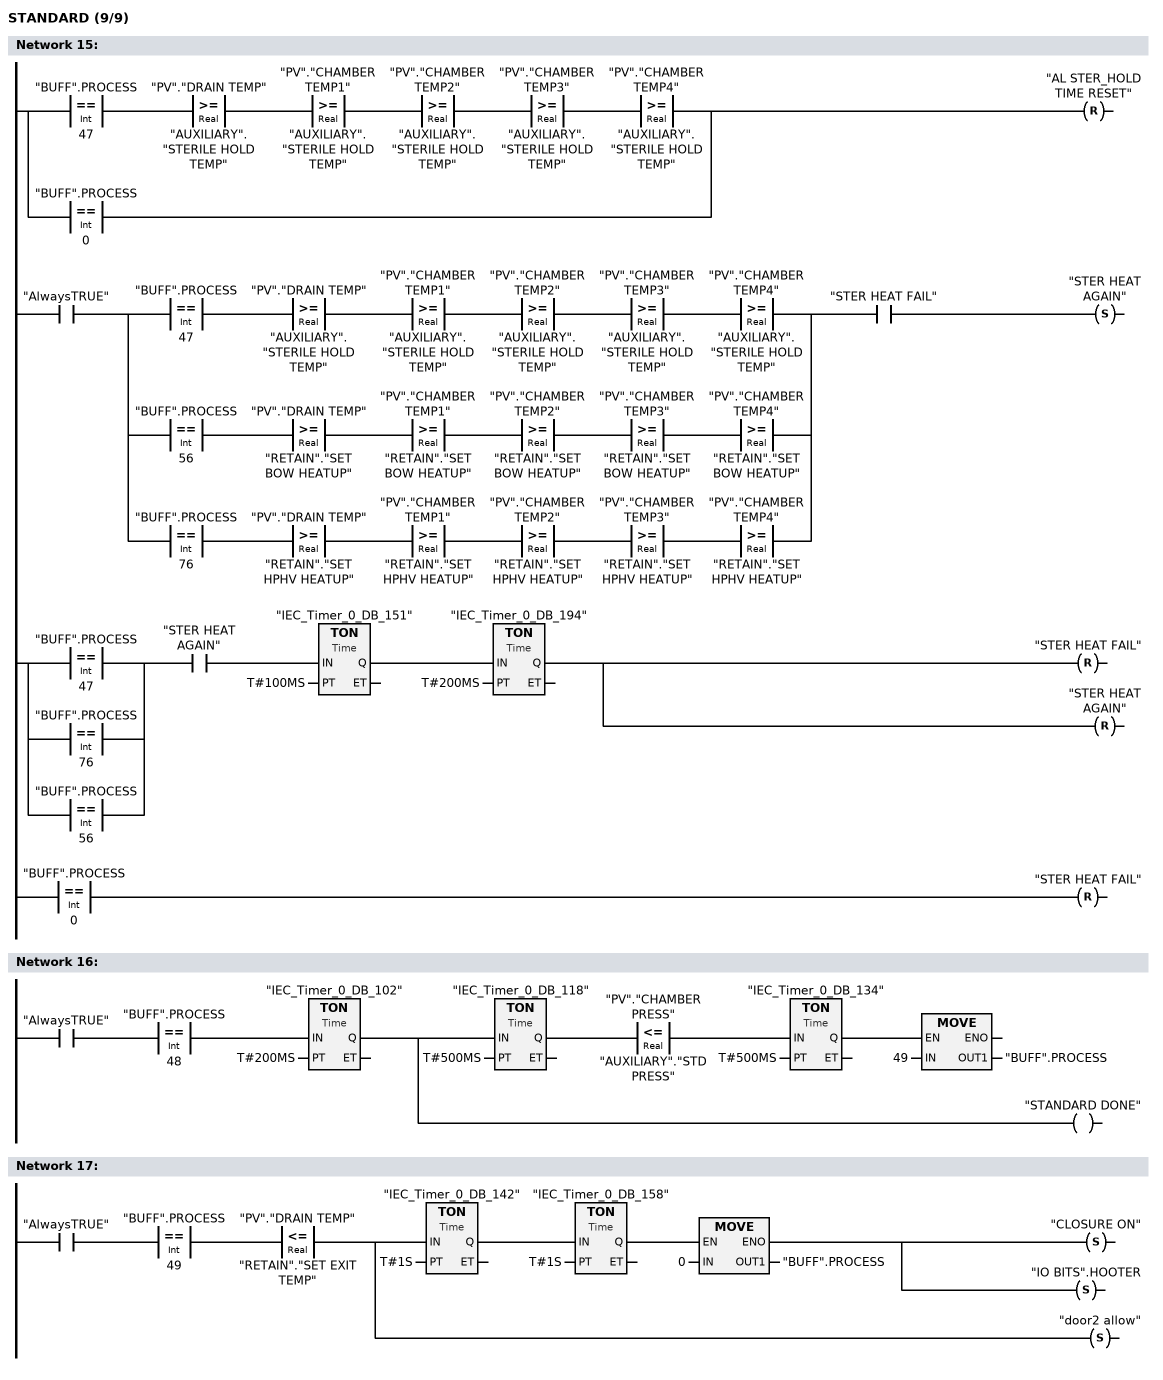
   RUNG wire#powerrail
      { S7_Templates := "SrcType := Int" } EQ_Contact(in1 := "BUFF".PROCESS, in2 := 47)
      { S7_Templates := "SrcType := Real" } GE_Contact(in1 := "PV"."DRAIN TEMP", in2 := "AUXILIARY"."STERILE HOLD TEMP")
      { S7_Templates := "SrcType := Real" } GE_Contact(in1 := "PV"."CHAMBER TEMP1", in2 := "AUXILIARY"."STERILE HOLD TEMP")
      { S7_Templates := "SrcType := Real" } GE_Contact(in1 := "PV"."CHAMBER TEMP2", in2 := "AUXILIARY"."STERILE HOLD TEMP")
      { S7_Templates := "SrcType := Real" } GE_Contact(in1 := "PV"."CHAMBER TEMP3", in2 := "AUXILIARY"."STERILE HOLD TEMP")
      { S7_Templates := "SrcType := Real" } GE_Contact(in1 := "PV"."CHAMBER TEMP4", in2 := "AUXILIARY"."STERILE HOLD TEMP")
      wire#w1
      R_Coil( "AL STER_HOLD TIME RESET" )
   END_RUNG
   RUNG wire#powerrail
      { S7_Templates := "SrcType := Int" } EQ_Contact(in1 := "BUFF".PROCESS, in2 := 0)
   END_RUNG wire#w1
   RUNG wire#powerrail
      Contact( "AlwaysTRUE" )
      wire#w2
      { S7_Templates := "SrcType := Int" } EQ_Contact(in1 := "BUFF".PROCESS, in2 := 47)
      { S7_Templates := "SrcType := Real" } GE_Contact(in1 := "PV"."DRAIN TEMP", in2 := "AUXILIARY"."STERILE HOLD TEMP")
      { S7_Templates := "SrcType := Real" } GE_Contact(in1 := "PV"."CHAMBER TEMP1", in2 := "AUXILIARY"."STERILE HOLD TEMP")
      { S7_Templates := "SrcType := Real" } GE_Contact(in1 := "PV"."CHAMBER TEMP2", in2 := "AUXILIARY"."STERILE HOLD TEMP")
      { S7_Templates := "SrcType := Real" } GE_Contact(in1 := "PV"."CHAMBER TEMP3", in2 := "AUXILIARY"."STERILE HOLD TEMP")
      { S7_Templates := "SrcType := Real" } GE_Contact(in1 := "PV"."CHAMBER TEMP4", in2 := "AUXILIARY"."STERILE HOLD TEMP")
      wire#w3
      Contact( "STER HEAT FAIL" )
      S_Coil( "STER HEAT AGAIN" )
   END_RUNG
   RUNG wire#w2
      { S7_Templates := "SrcType := Int" } EQ_Contact(in1 := "BUFF".PROCESS, in2 := 56)
      { S7_Templates := "SrcType := Real" } GE_Contact(in1 := "PV"."DRAIN TEMP", in2 := "RETAIN"."SET BOW HEATUP")
      { S7_Templates := "SrcType := Real" } GE_Contact(in1 := "PV"."CHAMBER TEMP1", in2 := "RETAIN"."SET BOW HEATUP")
      { S7_Templates := "SrcType := Real" } GE_Contact(in1 := "PV"."CHAMBER TEMP2", in2 := "RETAIN"."SET BOW HEATUP")
      { S7_Templates := "SrcType := Real" } GE_Contact(in1 := "PV"."CHAMBER TEMP3", in2 := "RETAIN"."SET BOW HEATUP")
      { S7_Templates := "SrcType := Real" } GE_Contact(in1 := "PV"."CHAMBER TEMP4", in2 := "RETAIN"."SET BOW HEATUP")
   END_RUNG wire#w3
   RUNG wire#w2
      { S7_Templates := "SrcType := Int" } EQ_Contact(in1 := "BUFF".PROCESS, in2 := 76)
      { S7_Templates := "SrcType := Real" } GE_Contact(in1 := "PV"."DRAIN TEMP", in2 := "RETAIN"."SET HPHV HEATUP")
      { S7_Templates := "SrcType := Real" } GE_Contact(in1 := "PV"."CHAMBER TEMP1", in2 := "RETAIN"."SET HPHV HEATUP")
      { S7_Templates := "SrcType := Real" } GE_Contact(in1 := "PV"."CHAMBER TEMP2", in2 := "RETAIN"."SET HPHV HEATUP")
      { S7_Templates := "SrcType := Real" } GE_Contact(in1 := "PV"."CHAMBER TEMP3", in2 := "RETAIN"."SET HPHV HEATUP")
      { S7_Templates := "SrcType := Real" } GE_Contact(in1 := "PV"."CHAMBER TEMP4", in2 := "RETAIN"."SET HPHV HEATUP")
   END_RUNG wire#w3
   RUNG wire#powerrail
      { S7_Templates := "SrcType := Int" } EQ_Contact(in1 := "BUFF".PROCESS, in2 := 47)
      wire#w4
      Contact( "STER HEAT AGAIN" )
      { S7_Templates := "time_type := Time" } "IEC_Timer_0_DB_151".TON(pt := T#100MS, et =>)
      { S7_Templates := "time_type := Time" } "IEC_Timer_0_DB_194".TON(pt := T#200MS, et =>)
      wire#w5
      R_Coil( "STER HEAT FAIL" )
   END_RUNG
   RUNG wire#powerrail
      { S7_Templates := "SrcType := Int" } EQ_Contact(in1 := "BUFF".PROCESS, in2 := 76)
   END_RUNG wire#w4
   RUNG wire#powerrail
      { S7_Templates := "SrcType := Int" } EQ_Contact(in1 := "BUFF".PROCESS, in2 := 56)
   END_RUNG wire#w4
   RUNG wire#w5
      R_Coil( "STER HEAT AGAIN" )
   END_RUNG
   RUNG wire#powerrail
      { S7_Templates := "SrcType := Int" } EQ_Contact(in1 := "BUFF".PROCESS, in2 := 0)
      R_Coil( "STER HEAT FAIL" )
   END_RUNG
   // the same network as SCL:
   IF (("BUFF".PROCESS = 47) AND ("PV"."DRAIN TEMP" >= "AUXILIARY"."STERILE HOLD TEMP") AND ("PV"."CHAMBER TEMP1" >= "AUXILIARY"."STERILE HOLD TEMP") AND ("PV"."CHAMBER TEMP2" >= "AUXILIARY"."STERILE HOLD TEMP") AND ("PV"."CHAMBER TEMP3" >= "AUXILIARY"."STERILE HOLD TEMP") AND ("PV"."CHAMBER TEMP4" >= "AUXILIARY"."STERILE HOLD TEMP")) OR ("BUFF".PROCESS = 0) THEN
       "AL STER_HOLD TIME RESET" := FALSE;
   END_IF;
   IF "AlwaysTRUE" AND ((("BUFF".PROCESS = 47) AND ("PV"."DRAIN TEMP" >= "AUXILIARY"."STERILE HOLD TEMP") AND ("PV"."CHAMBER TEMP1" >= "AUXILIARY"."STERILE HOLD TEMP") AND ("PV"."CHAMBER TEMP2" >= "AUXILIARY"."STERILE HOLD TEMP") AND ("PV"."CHAMBER TEMP3" >= "AUXILIARY"."STERILE HOLD TEMP") AND ("PV"."CHAMBER TEMP4" >= "AUXILIARY"."STERILE HOLD TEMP")) OR (("BUFF".PROCESS = 56) AND ("PV"."DRAIN TEMP" >= "RETAIN"."SET BOW HEATUP") AND ("PV"."CHAMBER TEMP1" >= "RETAIN"."SET BOW HEATUP") AND ("PV"."CHAMBER TEMP2" >= "RETAIN"."SET BOW HEATUP") AND ("PV"."CHAMBER TEMP3" >= "RETAIN"."SET BOW HEATUP") AND ("PV"."CHAMBER TEMP4" >= "RETAIN"."SET BOW HEATUP")) OR (("BUFF".PROCESS = 76) AND ("PV"."DRAIN TEMP" >= "RETAIN"."SET HPHV HEATUP") AND ("PV"."CHAMBER TEMP1" >= "RETAIN"."SET HPHV HEATUP") AND ("PV"."CHAMBER TEMP2" >= "RETAIN"."SET HPHV HEATUP") AND ("PV"."CHAMBER TEMP3" >= "RETAIN"."SET HPHV HEATUP") AND ("PV"."CHAMBER TEMP4" >= "RETAIN"."SET HPHV HEATUP"))) AND "STER HEAT FAIL" THEN
       "STER HEAT AGAIN" := TRUE;
   END_IF;
   "IEC_Timer_0_DB_151".TON(IN := (("BUFF".PROCESS = 47) OR ("BUFF".PROCESS = 76) OR ("BUFF".PROCESS = 56)) AND "STER HEAT AGAIN",
                           PT := T#100MS);
   "IEC_Timer_0_DB_194".TON(IN := "IEC_Timer_0_DB_151".Q, PT := T#200MS);
   IF "IEC_Timer_0_DB_194".Q THEN
       "STER HEAT FAIL" := FALSE;
       "STER HEAT AGAIN" := FALSE;
   END_IF;
   IF "BUFF".PROCESS = 0 THEN "STER HEAT FAIL" := FALSE; END_IF;
END_REGION

REGION Network 16
   RUNG wire#powerrail
      Contact( "AlwaysTRUE" )
      { S7_Templates := "SrcType := Int" } EQ_Contact(in1 := "BUFF".PROCESS, in2 := 48)
      { S7_Templates := "time_type := Time" } "IEC_Timer_0_DB_102".TON(pt := T#200MS, et =>)
      wire#w1
      { S7_Templates := "time_type := Time" } "IEC_Timer_0_DB_118".TON(pt := T#500MS, et =>)
      { S7_Templates := "SrcType := Real" } LE_Contact(in1 := "PV"."CHAMBER PRESS", in2 := "AUXILIARY"."STD PRESS")
      { S7_Templates := "time_type := Time" } "IEC_Timer_0_DB_134".TON(pt := T#500MS, et =>)
      Move(in := 49, out1 => "BUFF".PROCESS)
   END_RUNG
   RUNG wire#w1
      Coil( "STANDARD DONE" )
   END_RUNG
   // the same network as SCL:
   "IEC_Timer_0_DB_102".TON(IN := "AlwaysTRUE" AND ("BUFF".PROCESS = 48), PT := T#200MS);
   "IEC_Timer_0_DB_118".TON(IN := "IEC_Timer_0_DB_102".Q, PT := T#500MS);
   "IEC_Timer_0_DB_134".TON(IN := "IEC_Timer_0_DB_118".Q AND ("PV"."CHAMBER PRESS" <= "AUXILIARY"."STD PRESS"),
                           PT := T#500MS);
   IF "IEC_Timer_0_DB_134".Q THEN "BUFF".PROCESS := 49; END_IF;
   "STANDARD DONE" := "IEC_Timer_0_DB_102".Q;
END_REGION

REGION Network 17
   RUNG wire#powerrail
      Contact( "AlwaysTRUE" )
      { S7_Templates := "SrcType := Int" } EQ_Contact(in1 := "BUFF".PROCESS, in2 := 49)
      { S7_Templates := "SrcType := Real" } LE_Contact(in1 := "PV"."DRAIN TEMP", in2 := "RETAIN"."SET EXIT TEMP")
      wire#w1
      { S7_Templates := "time_type := Time" } "IEC_Timer_0_DB_142".TON(pt := T#1S, et =>)
      { S7_Templates := "time_type := Time" } "IEC_Timer_0_DB_158".TON(pt := T#1S, et =>)
      Move(in := 0, out1 => "BUFF".PROCESS)
      wire#w2
      S_Coil( "CLOSURE ON" )
   END_RUNG
   RUNG wire#w2
      S_Coil( "IO BITS".HOOTER )
   END_RUNG
   RUNG wire#w1
      S_Coil( "door2 allow" )
   END_RUNG
   // the same network as SCL:
   #_w1 := "AlwaysTRUE" AND ("BUFF".PROCESS = 49) AND ("PV"."DRAIN TEMP" <= "RETAIN"."SET EXIT TEMP");
   "IEC_Timer_0_DB_142".TON(IN := #_w1, PT := T#1S);
   "IEC_Timer_0_DB_158".TON(IN := "IEC_Timer_0_DB_142".Q, PT := T#1S);
   IF "IEC_Timer_0_DB_158".Q THEN
       "BUFF".PROCESS := 0;
       "CLOSURE ON" := TRUE;
       "IO BITS".HOOTER := TRUE;
   END_IF;
   IF #_w1 THEN "door2 allow" := TRUE; END_IF;
END_REGION
END_FUNCTION
